TYPE "UDT_MESLoadData"
VERSION : 0.1
   STRUCT
      PartTypeID : Int;
      RecipeNumber : Int;
      DMC : String[128];
      StationStatus : Int;
      ErrorCode : Int;
      StatusBits : DInt;
      CycleID : DInt;
      UnitPartTypeID : Int;
      Reserved : Array[1..8] of DInt;
   END_STRUCT;

END_TYPE

